{attribute 'GeneratedUsingTerminal: EJ3202-0000-0019'}
{attribute addProperty BoxType "EJ3202-0000-0019"}
{attribute addProperty Id "StatusAT %I*Status_F2CE6D917ValueAT %I*INT2"}
{attribute addProperty CRC "1245267073"}
{attribute addProperty Size "9"}
TYPE RTD_Inputs_Channel_4A394481 :
STRUCT
	{attribute addProperty Name "Status"}
	Status AT %I* : Status_F2CE6D91;
	{attribute addProperty Name "Value"}
	Value AT %I* : INT;
END_STRUCT
END_TYPE

(* stored: Version 1.2.0.0, ProductVersion 3.1.4024.9
   DUT RTD_Inputs_Channel_4A394481: Id {0e988451-7538-47f3-a3ac-125aaba77183} *)
